{attribute 'GeneratedUsingTerminal: KL3062'}
{attribute addProperty BoxType "KL3062"}
{attribute addProperty Id "Channel_1AT %Q*Channel_6576A6810Channel_2AT %Q*Channel_6576A6810"}
{attribute addProperty CRC "2957383796"}
{attribute addProperty Size "0"}
TYPE KL3062_B0461874 :
STRUCT
	{attribute addProperty Name "Channel_1"}
	Channel_1 : Channel_6576A681;
	{attribute addProperty Name "Channel_2"}
	Channel_2 : Channel_6576A681;
END_STRUCT
END_TYPE

(* stored: Version 1.2.0.0, ProductVersion 3.1.4024.9
   DUT KL3062_B0461874: Id {6a6abd8d-db2e-46d5-bd29-ab164af941c4} *)
